{attribute 'qualified_only'}
VAR_GLOBAL
	bRestartServer	: BOOL;
	bNewDataJustCame : BOOL;
END_VAR

(* stored: Version 1.1.0.1, ProductVersion 3.1.4024.9
   GVL GVL_MQTT_Common: Id {9ade70c4-4bb0-4835-91bf-df04d8dc4fad} *)
